PROGRAM Simulation
VAR
	fbT1				: TON;				//The temperature is decreased on a time dalay
	tCooling			: TIME := T#500MS;	//Cooling rate
	bReduceTemp			: BOOL;				//Signal for decreasing the temperature
	fbT2				: TON;				//The temperature is increased on a time delay
	tEnvironment		: TIME := T#2S;		//Delay time when the door is closed
	tEnvironmentDoorOpen: TIME := T#1S;		//Delay time when the door is open
	bRaiseTemp			: BOOL;				//Signal for increasing the temperature
	tImTemp				: TIME;				//Delay time
	nCounter			: INT;				//Iteration of the programm
END_VAR

//After the compressor has been activated due to fTempActual being too high, the temperature decreases.
//The temperature is decreased by 0.1°C per cycle after a delay of P_Cooling
IF GVL_VAR.bCompressor THEN
	fbT1(IN:= GVL_VAR.bCompressor, PT:= tCooling, Q=> bReduceTemp);
	IF bReduceTemp THEN
		GVL_VAR.fTempActual:= GVL_VAR.fTempActual-0.1;
		fbT1(IN:= FALSE);
	END_IF
END_IF

//If the door is open, the warming will occur faster; SEL chooses between tEnvironment or tEnvironmentDoorOpen
tImTemp:= SEL(GVL_VAR.bDoorOpen, tEnvironment, tEnvironmentDoorOpen);

//If the compressor is not in operation, then the cooling chamber will become warmer.
//The temperature is incremental by 0.1°C per cycle after a delay of tImTemp
fbT2(IN:= TRUE, PT:= tImTemp, Q=> bRaiseTemp);
IF bRaiseTemp THEN
	GVL_VAR.fTempActual:= GVL_VAR.fTempActual+0.1;
	fbT2(IN:= FALSE);
END_IF

nCounter := nCounter+1;

END_PROGRAM

(* stored: Version 1.1.0.1, ProductVersion 3.1.4024.4
   POU Simulation: Id {d80bc9b5-f326-44dc-8db6-962079a94870}, SpecialFunc None *)
